Staubli VAL3: start.pgx

program start()
begin
  movej(jHome,tTool,mNomSpeed)
  waitEndMove()
  movej(jAproachPiece,tTool,mNomSpeed)
  waitEndMove()
  movel(pGetObject,tTool,mNomSpeed)
  waitEndMove()
  open()
  waitEndMove()
  movej(jAproachPiece,tTool,mNomSpeed)
  waitEndMove()

end
